Fanuc KAREL source: kt00993.KL

-- PROVISIONAL review KL for V940-1; original PC SHA256 161d88f55276ab00aa6350eda579fc06e5fe3c41ee16ffc2fdb1f4e218908688
-- Incomplete behavior may be omitted. Consult companion uncertainty JSON. Do not deploy.
PROGRAM KT00993
%NOLOCKGROUP
VAR
  X : REAL
  Y : REAL
  Z : REAL
  W : REAL
  P : REAL
  R : REAL
-- UNRESOLVED_DECL P1 type=000106
-- UNRESOLVED_DECL P2 type=000106
-- UNRESOLVED_DECL CFG type=00001c
BEGIN
  -- V9_ZERO_TABLE_METADATA_HINT layout=0001; no indexed target words; source/name/runtime held
  -- UNRESOLVED_PC offsets 5-20; opcodes 2E,22,32,35
  -- UNRESOLVED_PC offsets 25-40; opcodes 2E,22,32,35
  -- UNRESOLVED_PC offsets 45-60; opcodes 2E,22,32,35
  -- UNRESOLVED_PC offsets 65-80; opcodes 2E,22,32,35
  -- UNRESOLVED_PC offsets 85-145; opcodes 27,27,49,7E,AD,22,22,22,22,22,22,22,76
  -- UNRESOLVED_PC offsets 150-154; opcodes 7F
END KT00993
